TYPE EtherCatDeviceStatuses :
STRUCT
	///Is the device in a healthy state?
	healthStatus: HealthStatus;
END_STRUCT
END_TYPE

(* stored: Version 1.1.0.1, ProductVersion 3.1.4019.2
   DUT EtherCatDeviceStatuses: Id {5caa72db-cb59-431a-89cf-1593c1c5b0b5} *)
